GLOBALCONSTANTS DefaultPool (* Global constants *)
  VAR_GLOBAL CONSTANT
    ISO_DESIGNATOR_WIDTH : UINT := 80;
    ISO_DESIGNATOR_HEIGHT : UINT := 80;
    ISO_MASK_SIZE : UINT := 480;
    ISO_VERSION_LABEL : STRING;
    MASK_WIDTH : UINT := 480;
    MASK_HEIGHT : UINT := 480;
    WorkingSet_0 : UINT := 0;
    DataMask_M1 : UINT := 1000;
    Container_Wheel_based_machine_speed : UINT := 3000;
    SoftKeyMask_S1 : UINT := 4000;
    OutputString_km_h : UINT := 11000;
    OutputString_m_s : UINT := 11001;
    OutputNumber_Wheel_based_machine_speed_km_h : UINT := 12000;
    OutputNumber_Wheel_based_machine_speed_m_s : UINT := 12001;
    Line_13000 : UINT := 13000;
    Tractor_wheel_slip : UINT := 20000;
    Battery_disconnect : UINT := 20001;
    Work_distance_travelled : UINT := 20002;
    NumberVariable_Wheel_based_machine_speed : UINT := 21000;
    FontAttributes_23000 : UINT := 23000;
    FontAttributes_23001 : UINT := 23001;
    LineAttributes_24000 : UINT := 24000;
  END_VAR
END_GLOBALCONSTANTS
